Staubli VAL3: refreshDynamic.pgx

program refreshDynamic()
begin
  // DO NOT CHANGE
  //
  // ADD HERE
  //
  call CycleRefresh()
  // print the instruction and the bar
  call printToShow()
  //
  // init
  use:bUseRefresh=false
  //
  // ADD HERE
  //
end
